FUNCTION_BLOCK fbGetUnixTime
VAR_INPUT
END_VAR
VAR_OUTPUT
END_VAR
VAR
    fbSystemTime : GETSYSTEMTIME;
    timeAsFileTime : T_FILETIME;
    timeAsSystemTime : TIMESTRUCT;
	timeAsDT : DT;
	timeAsULINT : ULINT;	
	
END_VAR

fbSystemTime(timeLoDW=>timeAsFileTime.dwLowDateTime, timeHiDW=>timeAsFileTime.dwHighDateTime);
timeAsSystemTime := FILETIME_TO_SYSTEMTIME(timeAsFileTime); //to get milliseconds
timeAsDT := FILETIME_TO_DT( timeAsFileTime );  //DT is only seconds, no MS component
unixTime := DT_TO_ULINT(timeAsDT) * 1000 + timeAsSystemTime.wMilliseconds; //global variable

END_FUNCTION_BLOCK

(* stored: Version 1.1.0.1, ProductVersion 3.1.0.36
   POU fbGetUnixTime: Id {622c589a-9bf2-409f-8b34-a1d4563a7481}, SpecialFunc None *)
